(* Some block comment for the struct *)
TYPE MyStruct :
STRUCT
	name : STRING;
	age : INT;
END_STRUCT
END_TYPE

(* stored: Version 1.1.0.1, ProductVersion 3.1.4024.11
   DUT MyStruct: Id {0ca2f239-e92f-475b-a644-4078618fc671} *)
